// TIA Portal project "032_100_FC-Programming_V14" (V14)

(* hardware
DEVICE "S71500/ET200MP station_1"  S7-1500 station
   slot 0: "Rail_0"  Rack  6ES7 590-1***0-0AA0
   slot 0: "PM 190W 120/230VAC"  PM 190W 120/230VAC  6EP1333-4BA00
   slot 1: "CPU1516F"  CPU 1516F-3 PN/DP  6ES7 516-3FN01-0AB0  V2.1
      slot 3: "CPU display_1"  6ES7591-1BA00-0AA0
   slot 2: "DI 32x24VDC HF_1"  DI 32x24VDC HF  6ES7 521-1BL00-0AB0  V2.1
   slot 3: "DQ 32x24VDC/0.5A HF_1"  DQ 32x24VDC/0.5A HF  6ES7 522-1BL01-0AB0  V1.0
   slot 4: "AI 8xU/I/RTD/TC ST_1"  AI 8xU/I/RTD/TC ST  6ES7 531-7KF00-0AB0  V2.1
   slot 5: "AQ 4xU/I ST_1"  AQ 4xU/I ST  6ES7 532-5HD00-0AB0  V2.1
*)

// ===== PLC "CPU1516F"  CPU 1516F-3 PN/DP =====

VAR_GLOBAL   // PLC tag table "Tag table_sorting station"
   "-A1" AT %I0.0 : Bool;   // return signal emergency stop ok (nc)
   "-K0" AT %I0.1 : Bool;   // main switch „ON“ (no)
   "-S0" AT %I0.2 : Bool;   // mode selector manual(0) / automatic(1)
   "-S1" AT %I0.3 : Bool;   // pushbutton automatic start (no)
   "-S2" AT %I0.4 : Bool;   // pushbutton automatic stop (nc)
   "-B1" AT %I0.5 : Bool;   // sensor cylinder -M4 retracted (no)
   "-B2" AT %I0.6 : Bool;   // sensor cylinder -M4 extended (nc)
   "-B3" AT %I0.7 : Bool;   // sensor motor -M1 actice (pulse signal for positioning) (no)
   "-B4" AT %I1.0 : Bool;   // sensor part at slide (no)
   "-B5" AT %I1.1 : Bool;   // sensor metal part (no)
   "-B6" AT %I1.2 : Bool;   // sensor part in front of cylinder -M4 (no)
   "-B7" AT %I1.3 : Bool;   // sensor part at end of conveyor (no)
   "-S3" AT %I1.4 : Bool;   // pushbutton manual mode conveyor –M1 forwards (no)
   "-S4" AT %I1.5 : Bool;   // pushbutton manual mode conveyor –M1 backwards (no)
   "-S5" AT %I1.6 : Bool;   // pushbutton manual mode cylinder -M4 retract (no)
   "-S6" AT %I1.7 : Bool;   // pushbutton manual mode cylinder -M4 extend (no)
   "-Q1" AT %Q0.0 : Bool;   // conveyor motor -M1 forwards fixed speed
   "-Q2" AT %Q0.1 : Bool;   // conveyor motor -M1 backwards fixed speed
   "-Q3" AT %Q0.2 : Bool;   // conveyor motor -M1 variable speed
   "-M2" AT %Q0.3 : Bool;   // cylinder -M4 retract
   "-M3" AT %Q0.4 : Bool;   // cylinder -M4 extend
   "-P1" AT %Q0.5 : Bool;   // display „main switch on“
   "-P2" AT %Q0.6 : Bool;   // display „manual mode“
   "-P3" AT %Q0.7 : Bool;   // display „automatic mode“
   "-P4" AT %Q1.0 : Bool;   // display „emergency stop activated“
   "-P5" AT %Q1.1 : Bool;   // display „automatic mode started“
   "-P6" AT %Q1.2 : Bool;   // display cylinder -M4 „retracted“
   "-P7" AT %Q1.3 : Bool;   // display cylinder -M4 „extended“
END_VAR

FUNCTION "MOTOR_MANUAL" : Void   // FC1, FBD
TITLE = Motor control in manual mode
{ S7_Optimized_Access := 'TRUE' }
VERSION : 0.1
// Conveyor motor in manual mode: If the pushbutton_manual_mode is operated, the enable conditions are granted and the safety shutoff is not activated the output
// Conveyor_motor_manual_mode is activated
   VAR_INPUT
      Manual_mode_active : Bool;   // Manual mode activated
      Pushbutton_manual_mode : Bool;   // Pushbutton manual mode conveyor on
      Enable_OK : Bool;   // All enable conditions OK
      Safety_shutoff_active : Bool;   // Safety shutoff active e.g. emergency stop operated
   END_VAR
   VAR_OUTPUT
      Conveyor_motor_manual_mode : Bool;   // Control of the conveyor motor in manual mode
   END_VAR
BEGIN

REGION Network 1: Control of the conveyor motor in manual mode
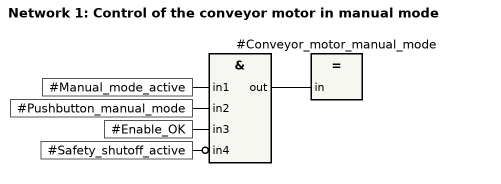
   #Conveyor_motor_manual_mode := #Manual_mode_active AND #Pushbutton_manual_mode AND #Enable_OK AND NOT #Safety_shutoff_active;
END_REGION
END_FUNCTION

FUNCTION "CYLINDER_MANUAL" : Void   // FC2, FBD
TITLE = Cylinder control in manual mode / Zylinderansteuerung Handbetrieb
{ S7_Optimized_Access := 'TRUE' }
VERSION : 0.1
// Cylinder in manual mode: If the pushbutton_manual_mode is operated, the enable conditions are granted and the safety shutoff is not activated the output
// Cylinder_manual_mode is activated
// Zylinder im Tippbetrieb: Der Ausgang Zylinder_Handbetrieb ist ein, solange der Taster_Tippbetrieb gedrückt, die Freigabe erteilt, und die Schutzabschaltung nicht aktiv ist.
   VAR_INPUT
      Manual_mode_active : Bool;   // Manual mode activated / Betriebsart Handbetrieb aktiviert
      Pushbutton_manual_mode : Bool;   // Pushbutton manual mode cylinder on / Taste um Zylinder im Tippbetrieb zu verfahren
      Enable_OK : Bool;   // All enable conditions OK / alle Freigabebedingungen erfüllt
      Safety_shutoff_active : Bool;   // Safety shutoff active e.g. emergency stop operated / Nothalt betätigt bzw. Schutzabschaltung aktiv
   END_VAR
   VAR_OUTPUT
      Cylinder_manual_mode : Bool;   // Control of the cylinder in manual mode / Zylinder im Handbetrieb ansteuern
   END_VAR
BEGIN

REGION Network 1: Control of the cylinder in manual mode / Zylinder im Tippbetrieb ansteuern
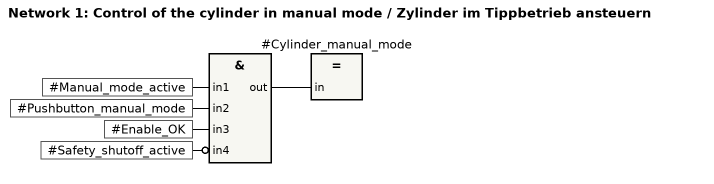
   #Cylinder_manual_mode := #Manual_mode_active AND #Pushbutton_manual_mode AND #Enable_OK AND NOT #Safety_shutoff_active;
END_REGION
END_FUNCTION

ORGANIZATION_BLOCK "Main"   // OB1, FBD, ProgramCycle
TITLE = "Main Program Sweep (Cycle)"
{ S7_Optimized_Access := 'TRUE' }
VERSION : 0.1
   VAR_INPUT
      Initial_Call : Bool;   // Initial call of this OB
      Remanence : Bool;   // =True, if remanent data are available
   END_VAR
BEGIN

REGION Network 1: Control conveyor motor forwards in manual mode
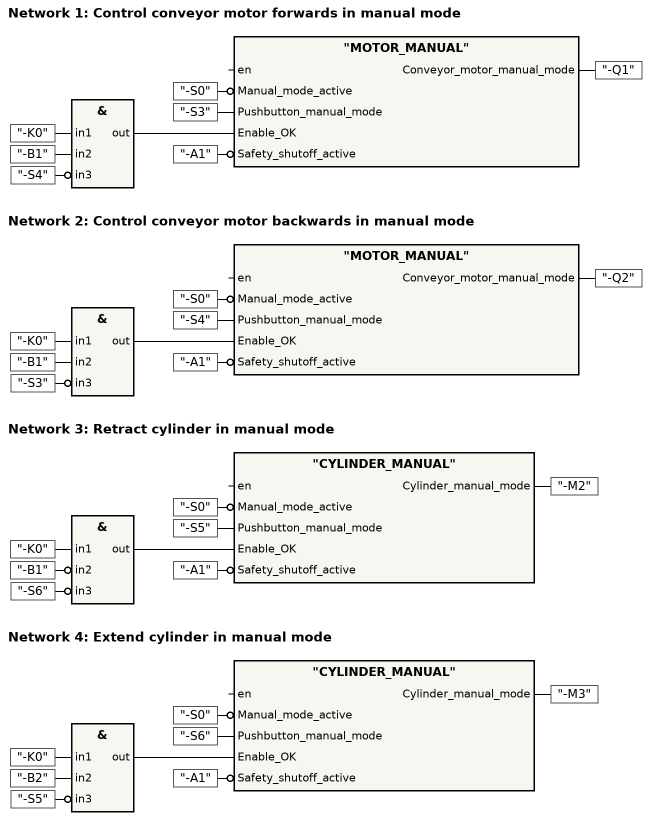
   "MOTOR_MANUAL"(Manual_mode_active := NOT "-S0",
                  Pushbutton_manual_mode := "-S3",
                  Enable_OK := "-K0" AND "-B1" AND NOT "-S4",
                  Safety_shutoff_active := NOT "-A1",
                  Conveyor_motor_manual_mode => "-Q1");
END_REGION

REGION Network 2: Control conveyor motor backwards in manual mode
   "MOTOR_MANUAL"(Manual_mode_active := NOT "-S0",
                  Pushbutton_manual_mode := "-S4",
                  Enable_OK := "-K0" AND "-B1" AND NOT "-S3",
                  Safety_shutoff_active := NOT "-A1",
                  Conveyor_motor_manual_mode => "-Q2");
END_REGION

REGION Network 3: Retract cylinder in manual mode
   "CYLINDER_MANUAL"(Manual_mode_active := NOT "-S0",
                     Pushbutton_manual_mode := "-S5",
                     Enable_OK := "-K0" AND NOT "-B1" AND NOT "-S6",
                     Safety_shutoff_active := NOT "-A1",
                     Cylinder_manual_mode => "-M2");
END_REGION

REGION Network 4: Extend cylinder in manual mode
   "CYLINDER_MANUAL"(Manual_mode_active := NOT "-S0",
                     Pushbutton_manual_mode := "-S6",
                     Enable_OK := "-K0" AND "-B2" AND NOT "-S5",
                     Safety_shutoff_active := NOT "-A1",
                     Cylinder_manual_mode => "-M3");
END_REGION
END_ORGANIZATION_BLOCK